// TwinCAT 3 PLC project technical_challenge
// ProgramVersion: 3.1.4024.0
// libraries:
//   Tc2_Standard, * (Beckhoff Automation GmbH)
//   Tc2_System, * (Beckhoff Automation GmbH)
//   Tc2_TcpIp, * (Beckhoff Automation GmbH)
//   Tc2_Utilities, * (Beckhoff Automation GmbH)
//   Tc3_Module, * (Beckhoff Automation GmbH)
// project tree:
//   DUTs/ E_State.TcDUT, OutputSignals.TcDUT, States.TcDUT, Timer.TcDUT
//   GVLs/ GVL.TcGVL
//   / PlcTask.TcTTO
//   POUs/ FB_TCPServer.TcPOU, MAIN.TcPOU, StateMachine.TcPOU
// real-time tasks:
//   TASK PlcTask: cycle T#10ms, priority 20, ADS port 350

CONFIGURATION technical_challenge
    RESOURCE PLC ON TwinCAT3
        TASK PlcTask(INTERVAL := T#10ms, PRIORITY := 20);
        PROGRAM MAIN WITH PlcTask : MAIN;
    END_RESOURCE
END_CONFIGURATION

// ---- DUTs/E_State.TcDUT
{attribute 'qualified_only'}
{attribute 'strict'}
TYPE E_State :
(
	STATE_1_Listen,
	STATE_2_Accept,
	STATE_3_Receive,
	STATE_4_Send
);
END_TYPE

// ---- DUTs/OutputSignals.TcDUT
TYPE OutputSignals :
STRUCT
	Motor1 : INT; // 1 is forward motion, -1 is backward motion, 0 standstill
	Motor2 : INT;  // 1 is counterclockwise rotation, -1 is clockwise rotation, 0 standstill
	GripperMotor : INT; // 1 is lift, -1 is lower, 0 is standstill
	Gripper : BOOL := TRUE; // TRUE when gripper open, FALSE when gripper is closed
END_STRUCT
END_TYPE

// ---- DUTs/States.TcDUT
{attribute 'qualified_only'}
{attribute 'strict'}
TYPE States :
(
	GRIPPER_OPEN := 0,
	ROTATE_DISC := 1,
	LINEAR_FW := 2,
	GRIPPER_LOWER := 3,
	GRIPPER_CLOSE := 4,
	GRIPPER_LIFT := 5,
	LINEAR_BW := 6
);
END_TYPE

// ---- DUTs/Timer.TcDUT
TYPE Timer :
STRUCT
	RotateDisc : TON;
	LinearFW : TON;
	GripperLower : TON;
	GripperOpen : TON;
	GripperClose: TON;
	GripperLift: TON;
	LinearBW : TON;
END_STRUCT
END_TYPE

// ---- GVLs/GVL.TcGVL
{attribute 'qualified_only'}
VAR_GLOBAL
	NUMBER_OF_SLOTS : INT := 6;
	SENSOR_POSITION_IN_DISC : INT := 4;
	
	ROTATE_DISC_TIME: TIME := T#1S;
	LINEAR_FW_TIME: TIME := T#1500MS;
	GRIPPER_LOWER_TIME: TIME := T#1S;
	GRIPPER_OPEN_TIME: TIME := T#500MS;
	GRIPPER_CLOSE_TIME: TIME := T#500MS;
	GRIPPER_LIFT_TIME: TIME := T#1S;
	GRIPPER_LINEAR_BW_TIME: TIME := T#1500MS;
END_VAR

// ---- POUs/MAIN.TcPOU
PROGRAM MAIN
VAR
	StateMachine: StateMachine;
	fbServer : FB_TCPServer;
	
	SrvNetId : STRING := '';
	ServerPort : UDINT := 9999;
	ServerAddress : STRING := '192.168.108.47';
	
	SResponse : STRING;
	SCommand : STRING;
	Received_data : STRING;
	
	Busy : BOOL;
	Error : BOOL;
	ErrId : UDINT;
	
	Toggle_Timer :TON;
	Mem_Bit AT %MX0.0 : BOOL :=FALSE;
END_VAR

StateMachine(OutputSignals=> );

fbServer(
	send_data:= SResponse, 
	NetId:= SrvNetId, 
	Server_Address:= ServerAddress, 
	Server_Port:= ServerPort, 
	Busy=> Busy, 
	Error=> Error, 
	Received_Data=> SCommand, 
	ErrId=> ErrId);

Toggle_Timer(IN:= NOT Toggle_Timer.Q, PT:= T#1000MS);
Mem_Bit := Toggle_Timer.ET > T#500MS;

SResponse := SCommand;

IF SCommand = 'bit_status' THEN
	IF Mem_Bit THEN
		SResponse := 'BIT ON';
	ELSE
		SResponse := 'BIT OFF';
	END_IF
END_IF

END_PROGRAM

// ---- POUs/StateMachine.TcPOU
FUNCTION_BLOCK StateMachine
VAR_INPUT
END_VAR
VAR_OUTPUT
	OutputSignals : OutputSignals;
END_VAR
VAR
	i : INT;
	state : States;
	Timer : Timer;
	Start: BOOL:=FALSE;
	CyclesCounter: CTU;
	TotalCyclesCounter : INT:=0;
	Reset : BOOL;
	CylinderInDisc : ARRAY[1..6] OF BOOL := [FALSE,5(TRUE)];
	Sensor: BOOL:= CylinderInDisc[GVL.SENSOR_POSITION_IN_DISC];
	PutCylinderInSlot6 : BOOL;
END_VAR

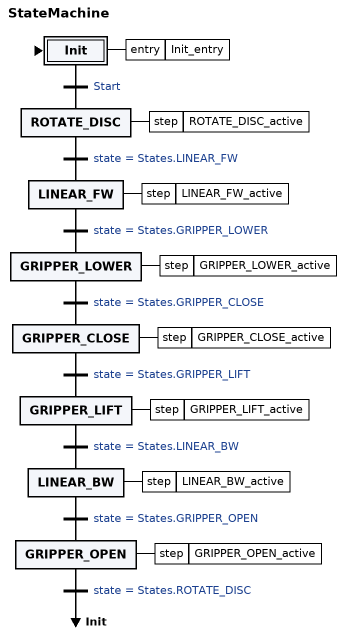
INITIAL_STEP Init:
    Init_entry(P1);  // entry action
END_STEP
TRANSITION FROM Init TO ROTATE_DISC
    := Start;
END_TRANSITION
STEP ROTATE_DISC:
    ROTATE_DISC_active(N);  // step action
END_STEP
TRANSITION FROM ROTATE_DISC TO LINEAR_FW
    := state = States.LINEAR_FW;
END_TRANSITION
STEP LINEAR_FW:
    LINEAR_FW_active(N);  // step action
END_STEP
TRANSITION FROM LINEAR_FW TO GRIPPER_LOWER
    := state = States.GRIPPER_LOWER;
END_TRANSITION
STEP GRIPPER_LOWER:
    GRIPPER_LOWER_active(N);  // step action
END_STEP
TRANSITION FROM GRIPPER_LOWER TO GRIPPER_CLOSE
    := state = States.GRIPPER_CLOSE;
END_TRANSITION
STEP GRIPPER_CLOSE:
    GRIPPER_CLOSE_active(N);  // step action
END_STEP
TRANSITION FROM GRIPPER_CLOSE TO GRIPPER_LIFT
    := state = States.GRIPPER_LIFT;
END_TRANSITION
STEP GRIPPER_LIFT:
    GRIPPER_LIFT_active(N);  // step action
END_STEP
TRANSITION FROM GRIPPER_LIFT TO LINEAR_BW
    := state = States.LINEAR_BW;
END_TRANSITION
STEP LINEAR_BW:
    LINEAR_BW_active(N);  // step action
END_STEP
TRANSITION FROM LINEAR_BW TO GRIPPER_OPEN
    := state = States.GRIPPER_OPEN;
END_TRANSITION
STEP GRIPPER_OPEN:
    GRIPPER_OPEN_active(N);  // step action
END_STEP
TRANSITION FROM GRIPPER_OPEN TO Init
    := state = States.ROTATE_DISC;
END_TRANSITION

ACTION GRIPPER_CLOSE_active:
Timer.GripperClose(IN:=TRUE, PT:=GVL.GRIPPER_CLOSE_TIME);

OutputSignals.Gripper := FALSE;

IF Timer.GripperClose.Q THEN
	state := States.GRIPPER_LIFT;
END_IF
END_ACTION

ACTION GRIPPER_LIFT_active:
Timer.GripperLift(IN:=TRUE, PT:=GVL.GRIPPER_LIFT_TIME);

OutputSignals.GripperMotor := BOOL_TO_INT(NOT Timer.GripperLift.Q);

IF Timer.GripperLift.Q THEN
	CylinderInDisc[1] := FALSE;
	state := States.LINEAR_BW;
END_IF
END_ACTION

ACTION GRIPPER_LOWER_active:
Timer.GripperLower(IN:=TRUE, PT:=GVL.GRIPPER_LOWER_TIME);

OutputSignals.GripperMotor := - BOOL_TO_INT(NOT Timer.GripperLower.Q);

IF Timer.GripperLower.Q THEN
	state := States.GRIPPER_CLOSE;
END_IF
END_ACTION

ACTION GRIPPER_OPEN_active:
Timer.GripperOpen(IN:=TRUE, PT:=GVL.GRIPPER_OPEN_TIME);

OutputSignals.Gripper := TRUE;

IF Timer.GripperOpen.Q THEN
	state := States.ROTATE_DISC;
END_IF
END_ACTION

ACTION Init_entry:
Sensor := CylinderInDisc[4];

Timer.RotateDisc(IN:=FALSE);
Timer.LinearFW(IN:=FALSE);
Timer.GripperLower(IN:=FALSE);
Timer.GripperOpen(IN:=FALSE);
Timer.GripperClose(IN:=FALSE);
Timer.GripperLift(IN:=FALSE);
Timer.LinearBW(IN:=FALSE);
Reset := CyclesCounter.Q;
CyclesCounter(CU:=state = States.ROTATE_DISC, RESET := Reset, PV:=INT_TO_WORD(GVL.NUMBER_OF_SLOTS));
END_ACTION

ACTION LINEAR_BW_active:
Timer.LinearBW(IN:=TRUE, PT:=GVL.LINEAR_FW_TIME);

OutputSignals.Motor1 := - BOOL_TO_INT(NOT Timer.LinearBW.Q);

IF Timer.LinearBW.Q THEN
	state := States.GRIPPER_OPEN;
END_IF
END_ACTION

ACTION LINEAR_FW_active:
Timer.LinearFW(IN:=TRUE, PT:=GVL.LINEAR_FW_TIME);

OutputSignals.Motor1 := BOOL_TO_INT(NOT Timer.LinearFW.Q);

IF Timer.LinearFW.Q THEN
	state := States.GRIPPER_LOWER;
END_IF
END_ACTION

ACTION ROTATE_DISC_active:
Timer.RotateDisc(IN:=TRUE, PT:=GVL.ROTATE_DISC_TIME);

OutputSignals.Motor2 := BOOL_TO_INT(NOT Timer.RotateDisc.Q);

IF Timer.RotateDisc.Q THEN
	Timer.RotateDisc(IN:=FALSE);
	FOR i:=1 TO 5 BY 1 DO
		CylinderInDisc[i] := CylinderInDisc[i+1];
	END_FOR;
	CylinderInDisc[6] := PutCylinderInSlot6;
	IF CylinderInDisc[1] THEN
		state := States.LINEAR_FW;
	END_IF	
END_IF
END_ACTION

END_FUNCTION_BLOCK

// ---- POUs/FB_TCPServer.TcPOU
FUNCTION_BLOCK FB_TCPServer
VAR_INPUT
	SendData : DWORD;
	ServerNetworkId : STRING;
	ServerAddress : STRING;
	ServerPort : UDINT;
END_VAR
VAR_OUTPUT
	Busy : BOOL;
	Error: BOOL;
	ReceivedData : DWORD;
	ErrorId : UDINT;
END_VAR
VAR
	SocketCloseAll : FB_SocketCloseAll := (sSrvNetID := '', tTimeout:=T#100S);
	SocketListen : FB_SocketListen := (bExecute := TRUE);
	SocketAccept : FB_SocketAccept;
	SocketSend : FB_SocketSend;
	SocketReceive : FB_SocketReceive;
	
	timer : TON := (PT:=T#500MS);
	
	HandleListener : T_HSOCKET;
	HandleSocket : T_HSOCKET;
	
	CloseAll : BOOL:= TRUE;
	ConnectionAccepted: BOOL;
	BufferData : STRING;
	Timeout : TIME := T#10S;
	
	state : E_State;	
END_VAR

IF CloseAll THEN
	CloseAll := FALSE;
	SocketCloseAll(bExecute :=TRUE);
ELSE
	SocketCloseAll(bExecute :=FALSE);
END_IF

timer(PT:=T#100MS);

SocketListen(
	sSrvNetId:= ServerNetworkId, 
	sLocalHost:= ServerAddress, 
	nLocalPort:= ServerPort, 
	bExecute:= , 
	tTimeout:= Timeout, 
	bBusy=> Busy, 
	bError=> Error, 
	nErrId=> ErrorId, 
	hListener=> HandleListener);
	
SocketAccept(
	sSrvNetId:= ServerNetworkId, 
	hListener:= HandleListener, 
	bExecute:= , 
	tTimeout:= Timeout, 
	bAccepted=> ConnectionAccepted, 
	bBusy=> Busy, 
	bError=> Error, 
	nErrId=> ErrorId, 
	hSocket=> HandleSocket);
	
SocketSend(
	sSrvNetId:= ServerNetworkId, 
	hSocket:= HandleSocket, 
	cbLen:= 4, 
	pSrc:= ADR(SendData), 
	bExecute:= , 
	tTimeout:= Timeout, 
	bBusy=> Busy, 
	bError=> Error, 
	nErrId=> ErrorId);

	
SocketReceive(
	sSrvNetId:= ServerNetworkId, 
	hSocket:= HandleSocket, 
	cbLen:= SIZEOF(BufferData), 
	pDest:= ADR(BufferData), 
	bExecute:= , 
	tTimeout:= Timeout, 
	bBusy=> Busy, 
	bError=> Error, 
	nErrId=> ErrorId, 
	nRecBytes=> );
	
	

CASE state OF
	E_State.STATE_1_Listen:
		SocketListen.bExecute := TRUE;
		state := E_State.STATE_2_Accept;
		
	E_State.STATE_2_Accept:
		SocketListen.bExecute := FALSE;
		IF NOT SocketListen.bBusy AND NOT SocketListen.bError THEN
			SocketAccept.bExecute := FALSE;
			timer.IN := TRUE;
			IF ConnectionAccepted THEN
				SocketReceive.bExecute := TRUE;
				state := E_State.STATE_3_Receive;
			ELSIF timer.Q THEN
				SocketAccept.bExecute := TRUE;
				timer.IN := FALSE;
			END_IF
		END_IF
		
	E_State.STATE_3_Receive:
		SocketReceive.bExecute := FALSE;
		IF NOT SocketReceive.bBusy AND NOT SocketReceive.bError THEN
			IF SocketReceive.nRecBytes = 0 THEN
				SocketReceive.bExecute := TRUE;
			ELSE
				MEMSET(
					destAddr := ADR(ReceivedData),
					fillByte := 0,
					n := SIZEOF(ReceivedData));
				MEMCPY (
					destAddr := ADR(ReceivedData),
					srcAddr := SocketReceive.pDest,
					n := SocketReceive.nRecBytes);
				
				SocketSend.bExecute := TRUE;
				state := E_State.STATE_4_Send;
			END_IF
		END_IF
		
	E_State.STATE_4_Send:
		SocketSend.bExecute := FALSE;
		IF NOT SocketSend.bBusy AND NOT SocketSend.bError THEN
			SocketReceive.bExecute := TRUE;
			state := E_State.STATE_3_Receive;
		END_IF
END_CASE

END_FUNCTION_BLOCK
